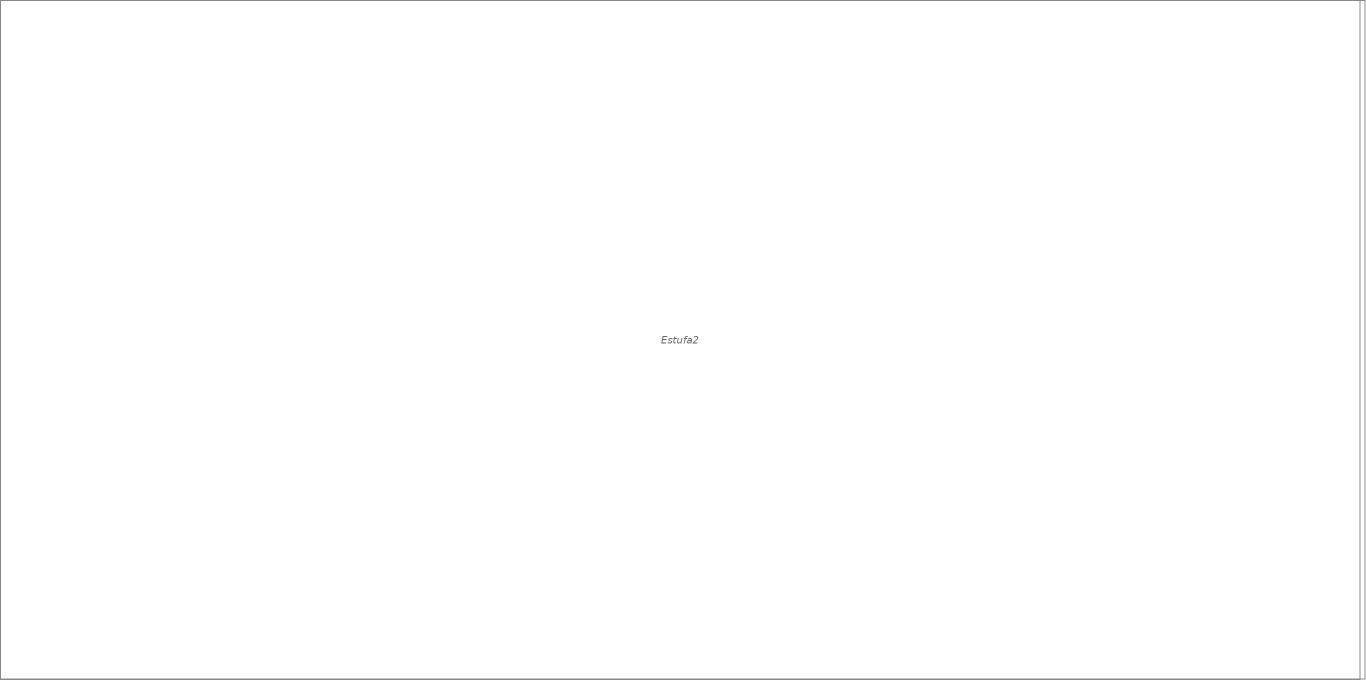
VISUALIZATION Aba_Estufa_2  // 1366x680
    TabControl (0,0 1360x680)
        shows Estufa2()
        shows Grafico_2()
        [0]: TabTitle=Dashboard
        [1]: TabTitle=Gráfico
END_VISUALIZATION

(* stored: Version 1.1.0.1, ProductVersion 3.1.4024.12
   Visu Aba_Estufa_2: Id {1af6530d-83da-4c61-8733-a2aaaf55dc69} *)
